FUNCTION_BLOCK FCC
  (* Version 1.0, 2006-08-11, Goran Cengic, Chalmers *)
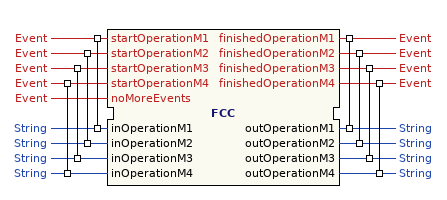
  EVENT_INPUT
    startOperationM1 WITH inOperationM1;
    startOperationM2 WITH inOperationM2;
    startOperationM3 WITH inOperationM3;
    startOperationM4 WITH inOperationM4;
    noMoreEvents;
  END_EVENT
  EVENT_OUTPUT
    finishedOperationM1 WITH outOperationM1;
    finishedOperationM2 WITH outOperationM2;
    finishedOperationM3 WITH outOperationM3;
    finishedOperationM4 WITH outOperationM4;
  END_EVENT
  VAR_INPUT
    inOperationM1 : String;
    inOperationM2 : String;
    inOperationM3 : String;
    inOperationM4 : String;
  END_VAR
  VAR_OUTPUT
    outOperationM1 : String;
    outOperationM2 : String;
    outOperationM3 : String;
    outOperationM4 : String;
  END_VAR
END_FUNCTION_BLOCK
